(* CODESYS project Codesys_ADT
   Author: Riley Duffy
   Company: Bosch Rexroth
   DefaultNamespace: ADT
   Description: Abstract Data Type Framework
   Title: ADT
   Version: 1.0.0

Project tree, tasks and I/O mapping:
  libraries: Standard, 3.5.18.0 (System)
  BoschSE_ADT.Sync
  commdata.all
  DUT/
    data type DummyType
    data type HashData
    data type PVoid
  DynamicInterfaces (Not Yet Tested)/
    interface iDynamicDataContainer: CopyToNew, EndResize, GetNew, GetNewPointer, StartResize
    interface iDynamicHashTable: Clear, Delete, isDeleted, isNewOccupied, isOccupied
  function block GettingStarted [ST]
  Interfaces/
    interface iCompare: Compare
    interface iDataContainer: Get, GetPointer, GetSize, Put
    interface iHash: Hash
    interface iHashTable: Clear, Delete, isDeleted, isOccupied
    interface iIterable: GetIterator, isBusy
    interface iIterator: Next, Size
    interface iList: Clear, CloseIterator, Find, Get, GetIterator, GetPointer, Insert, Pop, PushFront, Put, Remove
    interface iMap: Clear, Get, HasKey, Put, Remove
    interface iQueue: PopFront, PushBack, Size
    interface iStack: PopBack, PushBack, Size
  libADT.Sync
  function block License_And_Use [ST]
  POUs/
    ResizableMem (Not Fully Tested)/
      function block DynamicHashTable [ST]: Clear, Compare, CopyToNew, Delete, EndResize, Get, GetNew, GetNewPointer, GetPointer, GetSize, Hash, isDeleted, isNewOccupied, isOccupied, Put, StartResize
      function block DynamicList [ST]: Clear, CloseIterator, Find, Get, GetIterator, GetPointer, Insert, isBusy, Pop, PopBack, PopFront, PushBack, PushFront, Put, Remove, Resize, Size
      function block DynamicMap [ST]: Clear, Get, HasKey, Put, Remove, Resize
      function block DynamicQueue [ST]: PopFront, PushBack, Resize, Size
    StaticMem/
      function block HashTable [ST]: Clear, Compare, Delete, Get, GetPointer, GetSize, Hash, isDeleted, isOccupied, Put
      function block Iterator [ST]: GetIterator, isBusy, Next, Size
      function block List [ST]: Clear, CloseIterator, Find, Get, GetIterator, GetPointer, Insert, isBusy, Pop, PopBack, PopFront, PushBack, PushFront, Put, Remove, Size
      function block Map [ST]: Clear, Get, HasKey, Put, Remove
      function block Queue [ST]: PopFront, PushBack, Size
    Templates/
      function block TemplateDynamicContainer [ST]: CopyToNew, EndResize, FB_Exit, FB_Init, Get, GetNew, GetNewPointer, GetPointer, GetSize, Put, StartResize
      function block TemplateStaticDataContainer [ST]: Get, GetPointer, GetSize, Put
    Util/
      function block ADT_CompareString [ST]: Compare
      function block StringHash [ST]: Hash
  function GetLibVersion [ST]
  function GetLibVersionNumber [ST]
  function IsLibReleased [ST]
  function GetBooleanProperty [ST]
  function GetCompany [ST]
  function GetTextProperty2 [ST]
  function GetTextProperty [ST]
  function GetTitle [ST]
  function GetVersion [ST]
  function GetVersionProperty [ST]
*)

// DUT/DummyType
TYPE DummyType :
STRUCT
	dummy : BOOL; 
END_STRUCT
END_TYPE

// DUT/HashData
{attribute 'enable_dynamic_creation'}
TYPE HashData :
STRUCT
	isOccupied : BOOL; 
	isDeleted  : BOOL; 
END_STRUCT
END_TYPE

// DUT/PVoid
TYPE PVoid : __XWORD; END_TYPE

// GettingStarted
(*Use the Template container in POUs/Templates to quickly create your ADT Container. 
  Edit the _size and the DummyType to the size and type you want*)


FUNCTION_BLOCK GettingStarted
VAR_INPUT
END_VAR
VAR_OUTPUT
END_VAR
VAR
END_VAR

END_FUNCTION_BLOCK

// License_And_Use
(*
Copyright  2025 Riley Duffy

Permission is hereby granted, free of charge, to any person obtaining a copy of this software and associated documentation files
the “Software”), to deal in the Software without restriction, including without limitation the rights to use, copy, modify, merge,
publish, distribute, sublicense, and/or sell copies of the Software, and to permit persons to whom the Software is furnished to do so,
subject to the following conditions:

The above copyright notice and this permission notice shall be included in all copies or substantial portions of the Software.

THE SOFTWARE IS PROVIDED “AS IS”, WITHOUT WARRANTY OF ANY KIND, EXPRESS OR IMPLIED,
 INCLUDING BUT NOT LIMITED TO THE WARRANTIES OF MERCHANTABILITY, FITNESS FOR A PARTICULAR PURPOSE AND NONINFRINGEMENT.
 IN NO EVENT SHALL THE AUTHORS OR COPYRIGHT HOLDERS BE LIABLE FOR ANY CLAIM, DAMAGES OR OTHER LIABILITY,
 WHETHER IN AN ACTION OF CONTRACT, TORT OR OTHERWISE, ARISING FROM, OUT OF OR IN CONNECTION WITH THE SOFTWARE
 OR THE USE OR OTHER DEALINGS IN THE SOFTWARE.*)
FUNCTION_BLOCK License_And_Use
VAR_INPUT
END_VAR
VAR_OUTPUT
END_VAR
VAR
END_VAR

(*
Copyright  2025 Riley DUffy

Permission is hereby granted, free of charge, to any person obtaining a copy of this software and associated documentation files
(the “Software”), to deal in the Software without restriction, including without limitation the rights to use, copy, modify, merge,
publish, distribute, sublicense, and/or sell copies of the Software, and to permit persons to whom the Software is furnished to do so,
subject to the following conditions:

The above copyright notice and this permission notice shall be included in all copies or substantial portions of the Software.

THE SOFTWARE IS PROVIDED “AS IS”, WITHOUT WARRANTY OF ANY KIND, EXPRESS OR IMPLIED,
 INCLUDING BUT NOT LIMITED TO THE WARRANTIES OF MERCHANTABILITY, FITNESS FOR A PARTICULAR PURPOSE AND NONINFRINGEMENT.
 IN NO EVENT SHALL THE AUTHORS OR COPYRIGHT HOLDERS BE LIABLE FOR ANY CLAIM, DAMAGES OR OTHER LIABILITY,
 WHETHER IN AN ACTION OF CONTRACT, TORT OR OTHERWISE, ARISING FROM, OUT OF OR IN CONNECTION WITH THE SOFTWARE
 OR THE USE OR OTHER DEALINGS IN THE SOFTWARE.*)

END_FUNCTION_BLOCK

// DynamicInterfaces (Not Yet Tested)/iDynamicDataContainer
INTERFACE iDynamicDataContainer Extends iDataContainer;

METHOD CopyToNew : BOOL
VAR_INPUT
	indexOld :UDINT; 
	indexNew :UDINT; 
END_VAR
END_METHOD

METHOD EndResize : BOOL
VAR_INPUT
END_VAR
END_METHOD

METHOD GetNew : BOOL
VAR_INPUT
	index : UDINT;
	pData : PVoid;  
END_VAR
END_METHOD

METHOD GetNewPointer : PVoid
VAR_INPUT
	index : UDINT;
END_VAR
END_METHOD

METHOD StartResize : BOOL
VAR_INPUT
END_VAR
END_METHOD

END_INTERFACE

// Interfaces/iDataContainer
INTERFACE iDataContainer

METHOD Get : Bool
VAR_INPUT
	index : UDINT;
	pData : PVoid;  
END_VAR
END_METHOD

METHOD GetPointer : PVoid
VAR_INPUT
	index : UDINT;
END_VAR
END_METHOD

METHOD GetSize : UDINT
VAR_INPUT
END_VAR
END_METHOD

METHOD Put : Bool
VAR_INPUT
	index : UDINT; 
	pData : PVoid; 
END_VAR
END_METHOD

END_INTERFACE

// DynamicInterfaces (Not Yet Tested)/iDynamicHashTable
INTERFACE iDynamicHashTable EXTENDS iDynamicDataContainer,iCompare,iHash

METHOD Clear : Bool
VAR_INPUT
END_VAR
END_METHOD

METHOD Delete : Bool
VAR_INPUT
	index : UDINT; 
END_VAR
END_METHOD

METHOD isDeleted : Bool
VAR_INPUT
	index : UDINT;
END_VAR
END_METHOD

METHOD isNewOccupied : BOOL
VAR_INPUT
	index : UDINT; 
END_VAR
END_METHOD

METHOD isOccupied : bool
VAR_INPUT
	index : UDINT; 
END_VAR
END_METHOD

END_INTERFACE

// Interfaces/iCompare
INTERFACE iCompare

METHOD Compare : INT
VAR_INPUT
	pData1 : PVoid; 
	pData2 : PVoid; 
END_VAR
END_METHOD

END_INTERFACE

// Interfaces/iHash
INTERFACE iHash

METHOD Hash : LINT
VAR_INPUT
	pData : pVoid; 
END_VAR
END_METHOD

END_INTERFACE

// Interfaces/iHashTable
INTERFACE iHashTable EXTENDS iDataContainer,iCompare,iHash

METHOD Clear : Bool
VAR_INPUT
END_VAR
END_METHOD

METHOD Delete : Bool
VAR_INPUT
	index : UDINT; 
END_VAR
END_METHOD

METHOD isDeleted : Bool
VAR_INPUT
	index : UDINT;
END_VAR
END_METHOD

METHOD isOccupied : bool
VAR_INPUT
	index : UDINT; 
END_VAR
END_METHOD

END_INTERFACE

// Interfaces/iIterable
INTERFACE iIterable

METHOD GetIterator : iIterator
VAR_INPUT
END_VAR
END_METHOD

PROPERTY isBusy : BOOL
GET
END_GET
END_PROPERTY

END_INTERFACE

// Interfaces/iIterator
INTERFACE iIterator EXTENDS iIterable

METHOD Next : BOOL
VAR_INPUT
	pData : PVOID; 
END_VAR
END_METHOD

PROPERTY Size : UDINT
GET
END_GET
END_PROPERTY

END_INTERFACE

// Interfaces/iList
INTERFACE iList EXTENDS iStack,iQueue,iIterable

METHOD Clear : BOOL
VAR_INPUT
END_VAR
END_METHOD

METHOD CloseIterator : BOOL
VAR_INPUT
END_VAR
END_METHOD

METHOD Find : iIterator
VAR_INPUT
	Where : iCompare; 
	pData : PVoid; 
	indexList : iList;
END_VAR
END_METHOD

METHOD Get : BOOL
VAR_INPUT
	Index : UDINT; 
	pData : PVOID; 
END_VAR
END_METHOD

METHOD GetIterator : iIterator
VAR_INPUT
	
END_VAR
END_METHOD

METHOD GetPointer : Bool
VAR_INPUT
	Index	: UDINT;
END_VAR
VAR_OUTPUT
	pData : PVoid; 
END_VAR
END_METHOD

METHOD Insert : BOOL
VAR_INPUT
	StartIndex : UDINT; 
	Values   : iIterable; 
END_VAR
END_METHOD

METHOD Pop : BOOL
VAR_INPUT
	Index : UDINT; 
	pData : PVOID; 
END_VAR
END_METHOD

METHOD PushFront : BOOL
VAR_INPUT
	pData : PVOID; 
END_VAR
END_METHOD

METHOD Put : BOOL
VAR_INPUT
	Index : UDINT; 
	pData : PVoid; 
END_VAR
END_METHOD

METHOD Remove : BOOL
VAR_INPUT
	Where : iCompare; 
	pData : PVoid; 
END_VAR
END_METHOD

END_INTERFACE

// Interfaces/iStack
INTERFACE iStack

METHOD PopBack : Bool
VAR_INPUT
	pData : PVoid; 
END_VAR
END_METHOD

METHOD PushBack : Bool
VAR_INPUT
	pData : PVOID; 
END_VAR
END_METHOD

PROPERTY Size : UDINT
GET
END_GET
END_PROPERTY

END_INTERFACE

// Interfaces/iQueue
INTERFACE iQueue

METHOD PopFront : Bool
VAR_INPUT
	pData : PVoid; 
END_VAR
END_METHOD

METHOD PushBack : Bool
VAR_INPUT
	pData : PVOID; 
END_VAR
END_METHOD

PROPERTY Size : UDINT
GET
END_GET
END_PROPERTY

END_INTERFACE

// Interfaces/iMap
INTERFACE iMap

METHOD Clear : Bool
VAR_INPUT
END_VAR
END_METHOD

METHOD Get : Bool
VAR_INPUT
	pKey : pVoid; 
	pValue : pVoid; 
END_VAR
END_METHOD

METHOD HasKey : Bool
VAR_INPUT
	pKey : pVoid; 
END_VAR
END_METHOD

METHOD Put : Bool
VAR_INPUT
	pKey : pVoid; 
	pValue : pVoid; 
END_VAR
END_METHOD

METHOD Remove : Bool
VAR_INPUT
	pKey : pVoid; 
END_VAR
END_METHOD

END_INTERFACE

// GetLibVersion
// This function has been automatically generated from the project information.
FUNCTION GetLibVersion : VERSION
VAR_INPUT
	
END_VAR

GetLibVersion.uiMajor := 1;
GetLibVersion.uiMinor := 0;
GetLibVersion.uiServicePack := 0;
GetLibVersion.uiPatch := 65535;

END_FUNCTION

// GetLibVersionNumber
// This function has been automatically generated from the project information.
FUNCTION GetLibVersionNumber : DWORD
VAR_INPUT
	
END_VAR

GetLibVersionNumber := 16777471;

END_FUNCTION

// IsLibReleased
// This function has been automatically generated from the project information.
FUNCTION IsLibReleased : BOOL
VAR_INPUT
	
END_VAR

IsLibReleased := FALSE;

END_FUNCTION

// GetBooleanProperty
// This function has been automatically generated from the project information.
{attribute 'signature_flag' := '1073741824'}
{attribute 'register_in_runtime'}
FUNCTION GetBooleanProperty : BOOL
VAR_INPUT
	stKey: WSTRING;
END_VAR

IF stKey = "Released" THEN
	GetBooleanProperty := FALSE;
ELSE
	GetBooleanProperty := FALSE;
END_IF

END_FUNCTION

// GetCompany
// This function has been automatically generated from the project information.
{attribute 'signature_flag' := '1073741824'}
{attribute 'register_in_runtime'}
FUNCTION GetCompany : WSTRING
VAR_INPUT
	
END_VAR

GetCompany := "Bosch Rexroth";

END_FUNCTION

// GetTextProperty2
// This function has been automatically generated from the project information.
{attribute 'signature_flag' := '1073741824'}
{attribute 'register_in_runtime'}
FUNCTION GetTextProperty2 : POINTER TO WSTRING
VAR_INPUT
	stKey: WSTRING;
END_VAR

IF stKey = "Author" THEN
	GetTextProperty2 := ADR("Riley Duffy");
ELSIF stKey = "Company" THEN
	GetTextProperty2 := ADR("Bosch Rexroth");
ELSIF stKey = "DefaultNamespace" THEN
	GetTextProperty2 := ADR("ADT");
ELSIF stKey = "Description" THEN
	GetTextProperty2 := ADR("Abstract Data Type Framework");
ELSIF stKey = "Project" THEN
	GetTextProperty2 := ADR("BoschSE_ADT");
ELSIF stKey = "Title" THEN
	GetTextProperty2 := ADR("ADT");
ELSE
	GetTextProperty2 := ADR("");
END_IF

END_FUNCTION

// GetTextProperty
// This function has been automatically generated from the project information.
{attribute 'signature_flag' := '1073741824'}
{attribute 'register_in_runtime'}
FUNCTION GetTextProperty : WSTRING
VAR_INPUT
	stKey: WSTRING;
END_VAR

IF stKey = "Author" THEN
	GetTextProperty := "Riley Duffy";
ELSIF stKey = "Company" THEN
	GetTextProperty := "Bosch Rexroth";
ELSIF stKey = "DefaultNamespace" THEN
	GetTextProperty := "ADT";
ELSIF stKey = "Description" THEN
	GetTextProperty := "Abstract Data Type Framework";
ELSIF stKey = "Project" THEN
	GetTextProperty := "BoschSE_ADT";
ELSIF stKey = "Title" THEN
	GetTextProperty := "ADT";
ELSE
	GetTextProperty := "";
END_IF

END_FUNCTION

// GetTitle
// This function has been automatically generated from the project information.
{attribute 'signature_flag' := '1073741824'}
{attribute 'register_in_runtime'}
FUNCTION GetTitle : WSTRING
VAR_INPUT
	
END_VAR

GetTitle := "ADT";

END_FUNCTION

// GetVersion
// This function has been automatically generated from the project information.
{attribute 'signature_flag' := '1073741824'}
{attribute 'register_in_runtime'}
FUNCTION GetVersion : VERSION
VAR_INPUT
	
END_VAR

GetVersion.uiMajor := 1;
GetVersion.uiMinor := 0;
GetVersion.uiServicePack := 0;
GetVersion.uiPatch := 65535;

END_FUNCTION

// GetVersionProperty
// This function has been automatically generated from the project information.
{attribute 'signature_flag' := '1073741824'}
{attribute 'register_in_runtime'}
FUNCTION GetVersionProperty : VERSION
VAR_INPUT
	stKey: WSTRING;
END_VAR

IF stKey = "Version" THEN
	GetVersionProperty.uiMajor := 1;
	GetVersionProperty.uiMinor := 0;
	GetVersionProperty.uiServicePack := 0;
	GetVersionProperty.uiPatch := 65535;
ELSE
	GetVersionProperty.uiMajor := 0;
	GetVersionProperty.uiMinor := 0;
	GetVersionProperty.uiServicePack := 0;
	GetVersionProperty.uiPatch := 0;
END_IF

END_FUNCTION

// POUs/ResizableMem (Not Fully Tested)/DynamicHashTable
{attribute 'no_check'}
FUNCTION_BLOCK DynamicHashTable IMPLEMENTS iDynamicHashTable
VAR_INPUT
	KeyContainer : iDynamicDataContainer;
	HashDataContainer : iDynamicDataContainer;  
	Compareator : iCompare;
	Hasher      : iHash;  
END_VAR
VAR_OUTPUT
END_VAR
VAR
END_VAR

{attribute 'no_check'}
METHOD Clear : BOOL
VAR
	tHashData : HashData; 
	i : UDINT; 
END_VAR
tHashData.isDeleted := FALSE; 
tHashData.isOccupied := FALSE; 
FOR i := 0 TO HashDataContainer.GetSize() DO 
	HashDataContainer.Put(i,ADR(tHashData)); 
END_FOR
END_METHOD

METHOD Compare : INT
VAR_INPUT
	pData1	: PVoid;
	pData2	: PVoid;
END_VAR
Compare := Compareator.Compare(pData1,pData2);
END_METHOD

METHOD CopyToNew : BOOL
VAR_INPUT
	indexOld	: UDINT;
	indexNew	: UDINT;
END_VAR
KeyContainer.CopyToNew(indexOld,indexNew);
HashDataContainer.CopyToNew(indexOld,indexNew);
END_METHOD

METHOD Delete : BOOL
VAR_INPUT
	index	: UDINT;
END_VAR
VAR
	tHashData : HashData; 
END_VAR
tHashData.isDeleted := TRUE; 
tHashData.isOccupied := FALSE; 
HashDataContainer.Put(index,ADR(tHashData));
END_METHOD

METHOD EndResize : BOOL
KeyContainer.StartResize(); 
HashDataContainer.StartResize();
END_METHOD

METHOD Get : BOOL
VAR_INPUT
	index	: UDINT;
	pData	: PVoid;
END_VAR
KeyContainer.Get(index,pData);
END_METHOD

METHOD GetNew : BOOL
VAR_INPUT
	index : UDINT;
	pData : PVoid;  
END_VAR
KeyContainer.GetNew(index,pData);
END_METHOD

METHOD GetNewPointer : PVoid
VAR_INPUT
	index	: UDINT;
END_VAR
GetNewPointer := KeyContainer.GetNewPointer(index);
END_METHOD

METHOD GetPointer : PVoid
VAR_INPUT
	index	: UDINT;
END_VAR
GetPointer := KeyContainer.GetPointer(index);
END_METHOD

METHOD GetSize : UDINT
GetSize := KeyContainer.GetSize();
END_METHOD

METHOD Hash : LINT
VAR_INPUT
	pData	: pVoid;
END_VAR
Hash := Hasher.Hash(pData);
END_METHOD

METHOD isDeleted : BOOL
VAR_INPUT
	index	: UDINT;
END_VAR
VAR
	tHashData : HashData; 
END_VAR
HashDataContainer.Get(index,ADR(tHashData)); 
isDeleted := tHashData.isDeleted;
END_METHOD

METHOD isNewOccupied : BOOL
VAR_INPUT
	index: UDINT;
END_VAR
VAR
	tHashData: HashData;
END_VAR
HashDataContainer.GetNew(index,ADR(tHashData)); 
isNewOccupied:= tHashData.isOccupied;
END_METHOD

METHOD isOccupied : BOOL
VAR_INPUT
	index	: UDINT;
END_VAR
VAR
	tHashData : HashData; 
END_VAR
HashDataContainer.Get(index,ADR(tHashData)); 
isOccupied:= tHashData.isOccupied;
END_METHOD

METHOD Put : BOOL
VAR_INPUT
	index	: UDINT;
	pData	: PVoid;
END_VAR
VAR
	tHashData : HashData; 
END_VAR
tHashData.isDeleted := FALSE; 
tHashData.isOccupied := TRUE; 
HashDataContainer.Put(index,ADR(tHashData)); 
KeyContainer.Put(index,pData);
END_METHOD

METHOD StartResize : BOOL
KeyContainer.StartResize(); 
HashDataContainer.StartResize();
END_METHOD

END_FUNCTION_BLOCK

// POUs/ResizableMem (Not Fully Tested)/DynamicList
{attribute 'no_check'}
FUNCTION_BLOCK DynamicList IMPLEMENTS iList
VAR_INPUT
	DataContainer :  iDynamicDataContainer; 
END_VAR
VAR_OUTPUT
END_VAR
VAR
	_size : UDINT; 
	_iterator : Iterator; 
	_bIteratorOpened : BOOL; 
	_backingSize: UDINT;
	_front: UDINT;
END_VAR

METHOD Clear : BOOL
_size := 0;
END_METHOD

METHOD CloseIterator : BOOL
_bIteratorOpened := FALSE;
END_METHOD

{attribute 'no_check'}
METHOD Find : iIterator
VAR_INPUT
	Where	: iCompare;
	pData	: PVoid;
	indexList	: iList;
END_VAR
VAR
	_i : UDINT; 
	_index : UDINT; 
END_VAR
IF _backingSize = 0 THEN 
	_backingSize := DataContainer.GetSize(); 
END_IF
IF NOT _bIteratorOpened THEN 
	indexList.Clear(); 
	FOR _i := 0 TO _size -1 DO 
		IF Where.Compare(pData,DataContainer.GetPointer((_i + _front) MOD _backingSize)) = 0 THEN 
			_index := (_i + _front)MOD _backingSize; 
			indexList.PushBack(ADR(_index)); 
		END_IF
	END_FOR
	_iterator(bAll := FALSE, 
		  refList := THIS^, 
		  refIndex := indexList);
	Find := _iterator; 
	_bIteratorOpened := TRUE; 
ELSE
	Find := _iterator; 
END_IF;
END_METHOD

METHOD Get : BOOL
VAR_INPUT
	Index	: UDINT;
	pData	: PVOID;
END_VAR
IF _backingSize = 0 THEN 
	_backingSize := DataContainer.GetSize(); 
END_IF
IF Index < _size THEN 
	Get := DataContainer.Get((Index + _front) MOD _backingSize ,pData); 
ELSE 
	Get := FALSE; 
END_IF
END_METHOD

METHOD GetIterator : iIterator
IF NOT _bIteratorOpened THEN
	_bIteratorOpened := TRUE;  
	_iterator(bAll := TRUE, 
			refList := THIS^
			);
	GetIterator := _iterator; 
ELSE 
	GetIterator := _iterator; 
END_IF
END_METHOD

METHOD GetPointer : Bool
VAR_INPUT
	Index	: UDINT;
END_VAR
VAR_OUTPUT
	pData : PVoid; 
END_VAR
IF _backingSize = 0 THEN 
	_backingSize := DataContainer.GetSize(); 
END_IF
IF Index < _size THEN 
	pData := DataContainer.GetPointer((Index + _front) MOD _backingSize);
	GetPointer := TRUE; 
ELSE 
	GetPointer := FALSE; 
END_IF
END_METHOD

METHOD Insert : BOOL
VAR_INPUT
	StartIndex	: UDINT; //Start Index
	Values	: iIterable; //Iterable list of values to insert
END_VAR

VAR
	_i: UDINT;
	_index: UDINT;
	_destIndex: UDINT;
END_VAR
IF _backingSize = 0 THEN 
	_backingSize := DataContainer.GetSize(); 
END_IF
WHILE Values.GetIterator().Size >= (_backingSize - size) DO 
	_backingSize := THIS^.Resize();
END_WHILE
IF StartIndex <= _size AND NOT Values.GetIterator().isBusy THEN 
	IF StartIndex <> _size THEN 
		FOR _i := _size - 1  TO StartIndex BY - 1 DO
			_index := (_front + _i) MOD _backingSize; 
			_destIndex := (_index + Values.GetIterator().Size) MOD _backingSize; 
			DataContainer.Put(_destIndex,DataContainer.GetNewPointer(_index)); 
			IF _i = 0 THEN 
				EXIT; 
			END_IF
		END_FOR
	END_IF
	WHILE Values.GetIterator().Next(DataContainer.GetPointer((StartIndex + _front + _i) MOD _backingSize)) DO 
		_i := _i+1; 
		_size := _size + 1; 
	END_WHILE
	Insert := TRUE; 
ELSE 
	Insert := FALSE; 
END_IF
END_METHOD

PROPERTY isBusy : BOOL
GET
isBusy := _bIteratorOpened;
END_GET
END_PROPERTY

METHOD Pop : BOOL
VAR_INPUT
	Index	: UDINT;
	pData	: PVOID;
END_VAR

VAR
	_i: UDINT;
	_index: UDINT;
	_indexPlus1: UDINT;
END_VAR
IF _backingSize = 0 THEN 
	_backingSize := DataContainer.GetSize(); 
END_IF
IF Index < _size THEN 
	Pop := DataContainer.Get((Index + _front) MOD _backingSize,pData); 
	FOR _i := Index TO size -1 DO 
		_index := (_front + _i) MOD _backingSize; 
		_indexPlus1 := (_index + 1) MOD _backingSize; 
		DataContainer.Put(_index,DataContainer.GetPointer(_indexPlus1)); 
		IF _i = 0 THEN 
			EXIT; 
		END_IF
	END_FOR
	_size := _size - 1; 
ELSE 
	Pop := FALSE; 
END_IF
END_METHOD

METHOD PopBack : BOOL
VAR_INPUT
	pData	: PVoid;
END_VAR

VAR
END_VAR
IF _backingSize = 0 THEN 
	_backingSize := DataContainer.GetSize(); 
END_IF
IF _size > 0 THEN 
	PopBack := DataContainer.Get((_front + _size) MOD _backingSize ,pData); 
	_size := _size - 1; 
ELSE 
	PopBack := FALSE; 
END_IF
END_METHOD

METHOD PopFront : BOOL
VAR_INPUT
	pData	: PVoid;
END_VAR
IF _backingSize = 0 THEN 
	_backingSize := DataContainer.GetSize(); 
END_IF
IF _size > 0 THEN 
	PopFront := DataContainer.Get(_front,pData); 
	_size := _size - 1; 
	_front := (_front + 1) MOD _backingSize; 
ELSE 
	PopFront := FALSE; 
END_IF
END_METHOD

METHOD PushBack : BOOL
VAR_INPUT
	pData	: PVOID;
END_VAR
IF _backingSize = 0 THEN 
	_backingSize := DataContainer.GetSize(); 
END_IF
IF _size >= _backingSize THEN 
	_backingSize := THIS^.Resize(); 
END_IF
IF _size < _backingSize THEN 
	PushBack := DataContainer.Put((_front+_size) MOD _backingSize,pData); 
	_size := _size + 1;
ELSE 
	PushBack := FALSE; 
END_IF
END_METHOD

METHOD PushFront : BOOL
VAR_INPUT
	pData	: PVOID;
END_VAR
IF _backingSize = 0 THEN 
	_backingSize := DataContainer.GetSize(); 
END_IF
IF _size >= _backingSize THEN 
	_backingSize := THIS^.Resize(); 
END_IF
IF _size < _backingSize THEN 
	_front := _front -1; 
	IF _front >= _backingSize THEN 
		_front := _backingSize - 1; 
	END_IF
	PushFront := DataContainer.Put(_front,pData); 
	_size := _size + 1; 
ELSE 
	PushFront := FALSE; 
END_IF
END_METHOD

METHOD Put : BOOL
VAR_INPUT
	Index	: UDINT;
	pData	: PVoid;
END_VAR

VAR
	_i: UDINT;
	_index : UDINT;
	_indexSub1 : UDINT; 
END_VAR
IF _backingSize = 0 THEN 
	_backingSize := DataContainer.GetSize(); 
END_IF
IF _size >= _backingSize THEN 
	_backingSize := THIS^.Resize(); 
END_IF
IF _size < _backingSize AND Index <= _size THEN 
	IF Index <> _size THEN 
		FOR _i := _size  TO Index + 1 BY - 1 DO
			_index := (_front + _i) MOD _backingSize; 
			_indexSub1 := _index - 1; 
			IF (_indexSub1 >= _backingSize) THEN 
				_indexSub1 := _backingSize -1; 
			END_IF
			DataContainer.Put(_index,DataContainer.GetPointer(_indexSub1)); 
		END_FOR
	END_IF
	Put := DataContainer.Put((Index + _front)MOD _backingSize,pData); 
	_size := _size + 1; 
ELSE 
	Put := FALSE; 
END_IF
END_METHOD

METHOD Remove : BOOL
VAR_INPUT
	Where	: iCompare;
	pData   : PVoid; 
END_VAR

VAR
	_i: UDINT;
	_j: UDINT;
	_index : UDINT; 
	_indexPlus1 : UDINT; 
END_VAR
Remove := FALSE; 
IF _size = 0 THEN 
	RETURN; 
END_IF
FOR _i := 0 TO _size -1 DO 
	IF Where.Compare(pData,DataContainer.GetPointer((_i + _front) MOD _backingSize)) = 0 THEN 
		FOR _j := _i  TO _size-1 DO 
			_index := (_front + _j) MOD _backingSize; 
			_indexPlus1 := (_index + 1) MOD _backingSize; 
			DataContainer.Put(_index,DataContainer.GetPointer(_indexPlus1)); 
		END_FOR
		_size := _size - 1; 
		Remove := TRUE; 
		EXIT; 
	END_IF;
END_FOR
END_METHOD

METHOD PRIVATE Resize : UDINT
VAR_INPUT
END_VAR

VAR
	_i: UDINT;
END_VAR
DataContainer.StartResize(); 
FOR _i := 0 TO THIS^.Size -1 DO 
	DataContainer.CopyToNew((_front + _i) MOD _backingSize, _i); 
END_FOR
_front := 0; 
DataContainer.EndResize();
Resize := DataContainer.GetSize();
END_METHOD

PROPERTY Size : UDINT
GET
Size := _size;
END_GET
END_PROPERTY

END_FUNCTION_BLOCK

// POUs/StaticMem/Iterator
FUNCTION_BLOCK Iterator IMPLEMENTS iIterator
VAR_INPUT
	bAll : BOOL; 
	refList : iList; 
	refIndex :  iList; 
END_VAR
VAR_OUTPUT
END_VAR
VAR
	_index : UDINT; 
END_VAR

_index := 0;

METHOD GetIterator : iIterator
GetIterator := This^;
END_METHOD

PROPERTY isBusy : BOOL
GET
isBusy := _index <> 0;
END_GET
END_PROPERTY

{attribute 'no_check'}
METHOD Next : BOOL
VAR_INPUT
	pData	: PVOID;
END_VAR
VAR 
	pIndex : UDINT; 
END_VAR
IF bAll THEN 
	IF _index <refList.Size THEN 
		IF refList.Get(_index ,pData) THEN 
			_index := _index + 1; 
			Next := TRUE; 
		ELSE 
			_index := 0; 
			refList.CloseIterator(); 
			Next := FALSE; 
		END_IF
	ELSE 
		_index := 0; 
		refList.CloseIterator(); 
		Next := FALSE; 
	END_IF
ELSE 
	IF _index < refIndex.Size THEN 
		IF refIndex.Get(_index,ADR(pIndex)) THEN 
			refList.Get(pIndex,pData); 
			_index := _index + 1; 
			Next := TRUE; 
		ELSE 
			_index := 0; 
			refIndex.Clear(); 
			refList.CloseIterator(); 
			Next := FALSE; 
		END_IF
	ELSE 
		_index := 0; 
		refList.CloseIterator(); 
		Next := FALSE; 
	END_IF	
END_IF
END_METHOD

PROPERTY Size : UDINT
GET
IF bAll THEN 
	Size := refList.Size;
ELSE
	Size := refIndex.Size;
END_IF
END_GET
END_PROPERTY

END_FUNCTION_BLOCK

// POUs/StaticMem/List
{attribute 'no_check'}
FUNCTION_BLOCK List IMPLEMENTS iList
VAR_INPUT
	DataContainer : iDataContainer; 
END_VAR
VAR_OUTPUT
END_VAR
VAR
	_size : UDINT; 
	_iterator : Iterator; 
	_bIteratorOpened : BOOL; 
	_backingSize: UDINT;
	_front: UDINT;
END_VAR

METHOD Clear : BOOL
_size := 0;
END_METHOD

METHOD CloseIterator : BOOL
_bIteratorOpened := FALSE;
END_METHOD

{attribute 'no_check'}
METHOD Find : iIterator
VAR_INPUT
	Where	: iCompare;
	pData	: PVoid;
	indexList	: iList;
END_VAR
VAR
	_i : UDINT; 
	_index : UDINT; 
END_VAR
IF _backingSize = 0 THEN 
	_backingSize := DataContainer.GetSize(); 
END_IF
IF NOT _bIteratorOpened THEN 
	indexList.Clear(); 
	FOR _i := 0 TO _size -1 DO 
		IF Where.Compare(pData,DataContainer.GetPointer((_i + _front) MOD _backingSize)) = 0 THEN 
			_index := (_i + _front)MOD _backingSize; 
			indexList.PushBack(ADR(_index)); 
		END_IF
	END_FOR
	_iterator(bAll := FALSE, 
		  refList := THIS^, 
		  refIndex := indexList);
	Find := _iterator; 
	_bIteratorOpened := TRUE; 
ELSE
	Find := _iterator; 
END_IF;
END_METHOD

METHOD Get : BOOL
VAR_INPUT
	Index	: UDINT;
	pData	: PVOID;
END_VAR
IF _backingSize = 0 THEN 
	_backingSize := DataContainer.GetSize(); 
END_IF
IF Index < _size THEN 
	Get := DataContainer.Get((Index + _front) MOD _backingSize ,pData); 
ELSE 
	Get := FALSE; 
END_IF
END_METHOD

METHOD GetIterator : iIterator
IF NOT _bIteratorOpened THEN
	_bIteratorOpened := TRUE;  
	_iterator(bAll := TRUE, 
			refList := THIS^
			);
	GetIterator := _iterator; 
ELSE 
	GetIterator := _iterator; 
END_IF
END_METHOD

METHOD GetPointer : Bool
VAR_INPUT
	Index	: UDINT;
END_VAR
VAR_OUTPUT
	pData : PVoid; 
END_VAR
IF _backingSize = 0 THEN 
	_backingSize := DataContainer.GetSize(); 
END_IF
IF Index < _size THEN 
	pData := DataContainer.GetPointer((Index + _front) MOD _backingSize);
	GetPointer := TRUE; 
ELSE 
	GetPointer := FALSE; 
END_IF
END_METHOD

METHOD Insert : BOOL
VAR_INPUT
	StartIndex	: UDINT; //Index Insertion Starts At
	Values	: iIterable; //Iterable list of values to insert
END_VAR

VAR
	_i: UDINT;
	_index: UDINT;
	_destIndex: UDINT;
END_VAR
IF _backingSize = 0 THEN 
	_backingSize := DataContainer.GetSize(); 
END_IF
IF Values.GetIterator().Size < (_backingSize - size) AND StartIndex <= _size AND NOT Values.GetIterator().isBusy THEN 
	IF StartIndex <> _size THEN 
		FOR _i := _size - 1  TO StartIndex BY - 1 DO
			_index := (_front + _i) MOD _backingSize; 
			_destIndex := (_index + Values.GetIterator().Size) MOD _backingSize; 
			DataContainer.Put(_destIndex,DataContainer.GetPointer(_index)); 
			IF _i = 0 THEN 
				EXIT; 
			END_IF
		END_FOR
	END_IF
	WHILE Values.GetIterator().Next(DataContainer.GetPointer((StartIndex + _front + _i) MOD _backingSize)) DO 
		_i := _i+1; 
		_size := _size + 1; 
	END_WHILE
	Insert := TRUE; 
ELSE 
	Insert := FALSE; 
END_IF
END_METHOD

PROPERTY isBusy : BOOL
GET
isBusy := _bIteratorOpened;
END_GET
END_PROPERTY

METHOD Pop : BOOL
VAR_INPUT
	Index	: UDINT;
	pData	: PVOID;
END_VAR

VAR
	_i: UDINT;
	_index: UDINT;
	_indexPlus1: UDINT;
END_VAR
IF _backingSize = 0 THEN 
	_backingSize := DataContainer.GetSize(); 
END_IF
IF Index < _size THEN 
	Pop := DataContainer.Get((Index + _front) MOD _backingSize,pData); 
	FOR _i := Index TO size -1 DO 
		_index := (_front + _i) MOD _backingSize; 
		_indexPlus1 := (_index + 1) MOD _backingSize; 
		DataContainer.Put(_index,DataContainer.GetPointer(_indexPlus1)); 
		IF _i = 0 THEN 
			EXIT; 
		END_IF
	END_FOR
	_size := _size - 1; 
ELSE 
	Pop := FALSE; 
END_IF
END_METHOD

METHOD PopBack : BOOL
VAR_INPUT
	pData	: PVoid;
END_VAR

VAR
END_VAR
IF _backingSize = 0 THEN 
	_backingSize := DataContainer.GetSize(); 
END_IF
IF _size > 0 THEN 
	PopBack := DataContainer.Get((_front + _size) MOD _backingSize ,pData); 
	_size := _size - 1; 
ELSE 
	PopBack := FALSE; 
END_IF
END_METHOD

METHOD PopFront : BOOL
VAR_INPUT
	pData	: PVoid;
END_VAR
IF _backingSize = 0 THEN 
	_backingSize := DataContainer.GetSize(); 
END_IF
IF _size > 0 THEN 
	PopFront := DataContainer.Get(_front,pData); 
	_size := _size - 1; 
	_front := (_front + 1) MOD _backingSize; 
ELSE 
	PopFront := FALSE; 
END_IF
END_METHOD

METHOD PushBack : BOOL
VAR_INPUT
	pData	: PVOID;
END_VAR
IF _backingSize = 0 THEN 
	_backingSize := DataContainer.GetSize(); 
END_IF
IF _size < _backingSize THEN 
	PushBack := DataContainer.Put((_front+_size) MOD _backingSize,pData); 
	_size := _size + 1; 
ELSE 
	PushBack := FALSE; 
END_IF
END_METHOD

METHOD PushFront : BOOL
VAR_INPUT
	pData	: PVOID;
END_VAR
IF _backingSize = 0 THEN 
	_backingSize := DataContainer.GetSize(); 
END_IF
IF _size < _backingSize THEN 
	_front := _front -1; 
	IF _front >= _backingSize THEN 
		_front := _backingSize - 1; 
	END_IF
	PushFront := DataContainer.Put(_front,pData); 
	_size := _size + 1; 
ELSE 
	PushFront := FALSE; 
END_IF
END_METHOD

METHOD Put : BOOL
VAR_INPUT
	Index	: UDINT;
	pData	: PVoid;
END_VAR

VAR
	_i: UDINT;
	_index : UDINT;
	_indexSub1 : UDINT; 
END_VAR
IF _backingSize = 0 THEN 
	_backingSize := DataContainer.GetSize(); 
END_IF
IF _size < _backingSize AND Index <= _size THEN 
	IF Index <> _size THEN 
		FOR _i := _size  TO Index + 1 BY - 1 DO
			_index := (_front + _i) MOD _backingSize; 
			_indexSub1 := _index - 1; 
			IF (_indexSub1 >= _backingSize) THEN 
				_indexSub1 := _backingSize -1; 
			END_IF
			DataContainer.Put(_index,DataContainer.GetPointer(_indexSub1)); 
		END_FOR
	END_IF
	Put := DataContainer.Put((Index + _front)MOD _backingSize,pData); 
	_size := _size + 1; 
ELSE 
	Put := FALSE; 
END_IF
END_METHOD

METHOD Remove : BOOL
VAR_INPUT
	Where	: iCompare;
	pData   : PVoid; 
END_VAR

VAR
	_i: UDINT;
	_j: UDINT;
	_index : UDINT; 
	_indexPlus1 : UDINT; 
END_VAR
Remove := FALSE; 
IF _size = 0 THEN 
	RETURN; 
END_IF
FOR _i := 0 TO _size -1 DO 
	IF Where.Compare(pData,DataContainer.GetPointer((_i + _front) MOD _backingSize)) = 0 THEN 
		FOR _j := _i  TO _size-1 DO 
			_index := (_front + _j) MOD _backingSize; 
			_indexPlus1 := (_index + 1) MOD _backingSize; 
			DataContainer.Put(_index,DataContainer.GetPointer(_indexPlus1)); 
		END_FOR
		_size := _size - 1; 
		Remove := TRUE; 
		EXIT; 
	END_IF;
END_FOR
END_METHOD

PROPERTY Size : UDINT
GET
Size := _size;
END_GET
END_PROPERTY

END_FUNCTION_BLOCK

// POUs/ResizableMem (Not Fully Tested)/DynamicMap
{attribute 'no_check'}
FUNCTION_BLOCK DynamicMap IMPLEMENTS iMap
VAR_INPUT
	KeyContainer : iDynamicHashTable; 
	ValueContainer : iDynamicDataContainer; 
END_VAR
VAR_OUTPUT
END_VAR
VAR
	_backingSize : UDINT := 0;
	_size : DINT := 0;  
END_VAR

METHOD Clear : BOOL
KeyContainer.Clear();
END_METHOD

{attribute 'no_check'}
METHOD Get : BOOL
VAR_INPUT
	pKey	: pVoid;
	pValue	: pVoid;
END_VAR

VAR
	hash: LINT;
	index: UDINT;
	_i : UDINT; 
	_tIndex: UDINT;
END_VAR
Get := FALSE; 
IF(_backingSize = 0 ) THEN 
	_backingSize := KeyContainer.GetSize(); 
END_IF
hash :=  KeyContainer.Hash(pKey); 
index := LINT_TO_UDINT(hash MOD _backingSize); 
WHILE _i < _backingSize - 1 DO 
	_tIndex := (_i + index) MOD _backingSize; 
	IF NOT (KeyContainer.isOccupied(_tIndex) OR KeyContainer.isDeleted(_tIndex))THEN 
		EXIT; 
	END_IF
	IF KeyContainer.Compare(pKey, KeyContainer.GetPointer(_tIndex)) = 0 THEN 
		ValueContainer.Get(_tIndex,pValue); 
		Get := TRUE; 
		EXIT; 
	END_IF
	_i := _i+ 1; 
END_WHILE
END_METHOD

{attribute 'no_check'}
METHOD HasKey : BOOL
VAR_INPUT
	pKey : pVoid; 
END_VAR

VAR
	hash: LINT;
	index: UDINT;
	_i: UDINT;
	_tIndex: UDINT;
END_VAR
HasKey := FALSE; 
IF(_backingSize = 0 ) THEN 
	_backingSize := KeyContainer.GetSize(); 
END_IF
hash :=  KeyContainer.Hash(pKey); 
index := LINT_TO_UDINT(hash MOD _backingSize); 
WHILE _i < _backingSize - 1 DO 
	_tIndex := (_i + index) MOD _backingSize; 
	IF NOT (KeyContainer.isOccupied(_tIndex) OR KeyContainer.isDeleted(_tIndex))THEN 
		EXIT; 
	END_IF
	IF KeyContainer.Compare(pKey, KeyContainer.GetNewPointer(_tIndex)) = 0 THEN  
		HasKey := TRUE; 
		EXIT; 
	END_IF
	_i := _i+ 1; 
END_WHILE
END_METHOD

{attribute 'no_check'}
METHOD Put : BOOL
VAR_INPUT
	pKey	: pVoid;
	pValue	: pVoid;
END_VAR

VAR
	hash: LINT;
	index: UDINT;
	_i: UDINT;
	_tIndex: UDINT;
END_VAR
Put := FALSE; 
IF(_backingSize = 0 ) THEN 
	_backingSize := KeyContainer.GetSize(); 
END_IF
IF _size >= _backingSize THEN 
	_backingSize := resize(); 
END_IF
hash :=  KeyContainer.Hash(pKey); 
index := LINT_TO_UDINT(hash MOD _backingSize); 
WHILE _i < _backingSize - 1 DO 
	_tIndex := (_i + index) MOD _backingSize; 
	IF (KeyContainer.isOccupied(_tIndex)) THEN 
		IF KeyContainer.Compare(pKey, KeyContainer.GetNewPointer(_tIndex)) = 0 THEN 
			ValueContainer.Put(_tIndex,pValue); 
			PUT := TRUE; 
			EXIT;
		END_IF
	ELSE 
		ValueContainer.Put(_tIndex,pValue); 
		KeyContainer.Put(_tIndex,pKey); 
		PUT := TRUE; 
		_size := _size + 1; 
		EXIT;
	END_IF 	
	_i := _i + 1; 
END_WHILE
END_METHOD

{attribute 'no_check'}
METHOD Remove : BOOL
VAR_INPUT
	pKey	: pVoid;
END_VAR

VAR
	hash: LINT;
	index: UDINT;
	_i: UDINT;
	_tIndex: UDINT;
END_VAR
Remove := FALSE; 
IF(_backingSize = 0 ) THEN 
	_backingSize := KeyContainer.GetSize(); 
END_IF
hash :=  KeyContainer.Hash(pKey); 
index := LINT_TO_UDINT(hash MOD _backingSize); 
WHILE _i < _backingSize - 1 DO 
	_tIndex := (_i + index) MOD _backingSize; 
	IF NOT (KeyContainer.isOccupied(_tIndex) OR KeyContainer.isDeleted(_tIndex))THEN 
		EXIT; 
	END_IF
	IF KeyContainer.Compare(pKey, KeyContainer.GetNewPointer(_tIndex)) = 0 THEN 
		KeyContainer.Delete(_tIndex);  
		Remove := TRUE; 
		_size := _size -1; 
		EXIT; 
	END_IF
	_i := _i+ 1; 
END_WHILE
END_METHOD

METHOD PRIVATE Resize : UDINT
VAR_INPUT
END_VAR

VAR
	_i: UDINT;
	_newSize: UDINT;
	index: UDINT;
	hash: LINT;
	_tIndex: UDINT;
	_j: UINT;
END_VAR
ValueContainer.StartResize();
KeyContainer.StartResize(); 
_newSize := KeyContainer.GetSize(); 
FOR _i := 0 TO _backingSize DO 
	IF KeyContainer.isOccupied(_i) THEN 
		hash :=  KeyContainer.Hash(KeyContainer.GetPointer(_i)); 
		index := LINT_TO_UDINT(hash MOD _newSize); 
		_j := 0; 
		WHILE _j < _backingSize - 1 DO 
			_tIndex := (_j + index) MOD _newSize; 
			IF (KeyContainer.isNewOccupied(_tIndex)) THEN 
				IF KeyContainer.Compare(KeyContainer.GetPointer(_i), KeyContainer.GetNewPointer(_tIndex)) = 0 THEN 
					KeyContainer.CopyToNew(_i,_tindex); 
					ValueContainer.CopyToNew(_i,_tindex); 
					EXIT;
				END_IF
			ELSE 
				KeyContainer.CopyToNew(_i,_tindex); 
				ValueContainer.CopyToNew(_i,_tindex); 
				EXIT;
			END_IF 	
			_j := _j + 1; 
		END_WHILE
	END_IF
END_FOR
Resize := 2*_backingSize; 
ValueContainer.EndResize();
KeyContainer.EndResize();
END_METHOD

END_FUNCTION_BLOCK

// POUs/ResizableMem (Not Fully Tested)/DynamicQueue
{attribute 'no_check'}
FUNCTION_BLOCK DynamicQueue IMPLEMENTS iQueue
VAR_INPUT
	DataContainer : iDynamicDataContainer; 
END_VAR
VAR_OUTPUT
END_VAR
VAR
	_size : UDINT; 
	_front: UDINT; 
	_backingSize : UDINT := 0; 
END_VAR

METHOD PopFront : BOOL
VAR_INPUT
	pData: PVoid;
END_VAR
IF _backingSize = 0 THEN 
	_backingSize := DataContainer.GetSize(); 
END_IF
IF _size > 0 THEN 
	PopFront := DataContainer.Get(_front,pData); 
	_size := _size - 1; 
	_front := (_front + 1) MOD _backingSize; 
ELSE 
	PopFront := FALSE; 
END_IF
END_METHOD

METHOD PushBack : BOOL
VAR_INPUT
	pData : pVoid; 
END_VAR
IF _backingSize = 0 THEN 
	_backingSize := DataContainer.GetSize(); 
END_IF
IF _size = _backingSize THEN 
	_backingSize := resize(); 
END_IF
IF _size < _backingSize THEN 
	PushBack := DataContainer.Put((_front+_size) MOD _backingSize,pData); 
	_size := _size + 1; 
ELSE 
	PushBack := FALSE; 
END_IF
END_METHOD

METHOD PRIVATE Resize : UDINT
VAR_INPUT
END_VAR

VAR
	_i: UDINT;
END_VAR
DataContainer.StartResize(); 
FOR _i := 0 TO THIS^.Size DO 
	DataContainer.CopyToNew((_front + _i) MOD _size, _i); 
END_FOR
_front := 0; 
DataContainer.EndResize();
Resize := DataContainer.GetSize();
END_METHOD

PROPERTY Size : UDINT
GET
Size := _size;
END_GET
END_PROPERTY

END_FUNCTION_BLOCK

// POUs/StaticMem/HashTable
{attribute 'no_check'}
FUNCTION_BLOCK HashTable IMPLEMENTS iHashTable
VAR_INPUT
	KeyContainer : iDataContainer;
	HashDataContainer : iDataContainer;  
	Compareator : iCompare;
	Hasher      : iHash;  
END_VAR
VAR_OUTPUT
END_VAR
VAR
END_VAR

{attribute 'no_check'}
METHOD Clear : BOOL
VAR
	tHashData : HashData; 
	i : UDINT; 
END_VAR
tHashData.isDeleted := FALSE; 
tHashData.isOccupied := FALSE; 
FOR i := 0 TO HashDataContainer.GetSize() DO 
	HashDataContainer.Put(i,ADR(tHashData)); 
END_FOR
END_METHOD

METHOD Compare : INT
VAR_INPUT
	pData1	: PVoid;
	pData2	: PVoid;
END_VAR
Compare := Compareator.Compare(pData1,pData2);
END_METHOD

METHOD Delete : BOOL
VAR_INPUT
	index	: UDINT;
END_VAR
VAR
	tHashData : HashData; 
END_VAR
tHashData.isDeleted := TRUE; 
tHashData.isOccupied := FALSE; 
HashDataContainer.Put(index,ADR(tHashData));
END_METHOD

METHOD Get : BOOL
VAR_INPUT
	index	: UDINT;
	pData	: PVoid;
END_VAR
KeyContainer.Get(index,pData);
END_METHOD

METHOD GetPointer : PVoid
VAR_INPUT
	index	: UDINT;
END_VAR
GetPointer := KeyContainer.GetPointer(index);
END_METHOD

METHOD GetSize : UDINT
GetSize := KeyContainer.GetSize();
END_METHOD

METHOD Hash : LINT
VAR_INPUT
	pData	: pVoid;
END_VAR
Hash := Hasher.Hash(pData);
END_METHOD

METHOD isDeleted : BOOL
VAR_INPUT
	index	: UDINT;
END_VAR
VAR
	tHashData : HashData; 
END_VAR
HashDataContainer.Get(index,ADR(tHashData)); 
isDeleted := tHashData.isDeleted;
END_METHOD

METHOD isOccupied : BOOL
VAR_INPUT
	index	: UDINT;
END_VAR
VAR
	tHashData : HashData; 
END_VAR
HashDataContainer.Get(index,ADR(tHashData)); 
isOccupied:= tHashData.isOccupied;
END_METHOD

METHOD Put : BOOL
VAR_INPUT
	index	: UDINT;
	pData	: PVoid;
END_VAR
VAR
	tHashData : HashData; 
END_VAR
tHashData.isDeleted := FALSE; 
tHashData.isOccupied := TRUE; 
HashDataContainer.Put(index,ADR(tHashData)); 
KeyContainer.Put(index,pData);
END_METHOD

END_FUNCTION_BLOCK

// POUs/StaticMem/Map
{attribute 'no_check'}
FUNCTION_BLOCK Map IMPLEMENTS iMap
VAR_INPUT
	KeyContainer : iHashTable; 
	ValueContainer : iDataContainer; 
END_VAR
VAR_OUTPUT
END_VAR
VAR
	_backingSize : UDINT := 0; 
END_VAR

METHOD Clear : BOOL
KeyContainer.Clear();
END_METHOD

{attribute 'no_check'}
METHOD Get : BOOL
VAR_INPUT
	pKey	: pVoid;
	pValue	: pVoid;
END_VAR

VAR
	hash: LINT;
	index: UDINT;
	_i : UDINT; 
	_tIndex: UDINT;
END_VAR
Get := FALSE; 
IF(_backingSize = 0 ) THEN 
	_backingSize := KeyContainer.GetSize(); 
END_IF
hash :=  KeyContainer.Hash(pKey); 
index := LINT_TO_UDINT(hash MOD _backingSize); 
WHILE _i < _backingSize - 1 DO 
	_tIndex := (_i + index) MOD _backingSize; 
	IF NOT (KeyContainer.isOccupied(_tIndex) OR KeyContainer.isDeleted(_tIndex))THEN 
		EXIT; 
	END_IF
	IF KeyContainer.Compare(pKey, KeyContainer.GetPointer(_tIndex)) = 0 THEN 
		ValueContainer.Get(_tIndex,pValue); 
		Get := TRUE; 
		EXIT; 
	END_IF
	_i := _i+ 1; 
END_WHILE
END_METHOD

{attribute 'no_check'}
METHOD HasKey : BOOL
VAR_INPUT
	pKey : pVoid; 
END_VAR

VAR
	hash: LINT;
	index: UDINT;
	_i: UDINT;
	_tIndex: UDINT;
END_VAR
HasKey := FALSE; 
IF(_backingSize = 0 ) THEN 
	_backingSize := KeyContainer.GetSize(); 
END_IF
hash :=  KeyContainer.Hash(pKey); 
index := LINT_TO_UDINT(hash MOD _backingSize); 
WHILE _i < _backingSize - 1 DO 
	_tIndex := (_i + index) MOD _backingSize; 
	IF NOT (KeyContainer.isOccupied(_tIndex) OR KeyContainer.isDeleted(_tIndex))THEN 
		EXIT; 
	END_IF
	IF KeyContainer.Compare(pKey, KeyContainer.GetPointer(_tIndex)) = 0 THEN  
		HasKey := TRUE; 
		EXIT; 
	END_IF
	_i := _i+ 1; 
END_WHILE
END_METHOD

{attribute 'no_check'}
METHOD Put : BOOL
VAR_INPUT
	pKey	: pVoid;
	pValue	: pVoid;
END_VAR

VAR
	hash: LINT;
	index: UDINT;
	_i: UDINT;
	_tIndex: UDINT;
END_VAR
Put := FALSE; 
IF(_backingSize = 0 ) THEN 
	_backingSize := KeyContainer.GetSize(); 
END_IF
hash :=  KeyContainer.Hash(pKey); 
index := LINT_TO_UDINT(hash MOD _backingSize); 
WHILE _i < _backingSize - 1 DO 
	_tIndex := (_i + index) MOD _backingSize; 
	IF (KeyContainer.isOccupied(_tIndex)) THEN 
		IF KeyContainer.Compare(pKey, KeyContainer.GetPointer(_tIndex)) = 0 THEN 
			ValueContainer.Put(_tIndex,pValue); 
			PUT := TRUE; 
			EXIT;
		END_IF
	ELSE 
		ValueContainer.Put(_tIndex,pValue); 
		KeyContainer.Put(_tIndex,pKey); 
		PUT := TRUE; 
		EXIT;
	END_IF 	
	_i := _i + 1; 
END_WHILE
END_METHOD

{attribute 'no_check'}
METHOD Remove : BOOL
VAR_INPUT
	pKey	: pVoid;
END_VAR

VAR
	hash: LINT;
	index: UDINT;
	_i: UDINT;
	_tIndex: UDINT;
END_VAR
Remove := FALSE; 
IF(_backingSize = 0 ) THEN 
	_backingSize := KeyContainer.GetSize(); 
END_IF
hash :=  KeyContainer.Hash(pKey); 
index := LINT_TO_UDINT(hash MOD _backingSize); 
WHILE _i < _backingSize - 1 DO 
	_tIndex := (_i + index) MOD _backingSize; 
	IF NOT (KeyContainer.isOccupied(_tIndex) OR KeyContainer.isDeleted(_tIndex))THEN 
		EXIT; 
	END_IF
	IF KeyContainer.Compare(pKey, KeyContainer.GetPointer(_tIndex)) = 0 THEN 
		KeyContainer.Delete(_tIndex);  
		Remove := TRUE; 
		EXIT; 
	END_IF
	_i := _i+ 1; 
END_WHILE
END_METHOD

END_FUNCTION_BLOCK

// POUs/StaticMem/Queue
{attribute 'no_check'}
FUNCTION_BLOCK Queue IMPLEMENTS iQueue
VAR_INPUT
	DataContainer : iDataContainer; 
END_VAR
VAR_OUTPUT
END_VAR
VAR
	_size : UDINT; 
	_front: UDINT; 
	_backingSize : UDINT := 0; 
END_VAR

METHOD PopFront : BOOL
VAR_INPUT
	pData: PVoid;
END_VAR
IF _backingSize = 0 THEN 
	_backingSize := DataContainer.GetSize(); 
END_IF
IF _size > 0 THEN 
	PopFront := DataContainer.Get(_front,pData); 
	_size := _size - 1; 
	_front := (_front + 1) MOD _backingSize; 
ELSE 
	PopFront := FALSE; 
END_IF
END_METHOD

METHOD PushBack : BOOL
VAR_INPUT
	pData : pVoid; 
END_VAR
IF _backingSize = 0 THEN 
	_backingSize := DataContainer.GetSize(); 
END_IF
IF _size < _backingSize THEN 
	PushBack := DataContainer.Put((_front+_size) MOD _backingSize,pData); 
	_size := _size + 1; 
ELSE 
	PushBack := FALSE; 
END_IF
END_METHOD

PROPERTY Size : UDINT
GET
Size := _size;
END_GET
END_PROPERTY

END_FUNCTION_BLOCK

// POUs/Templates/TemplateDynamicContainer
FUNCTION_BLOCK TemplateDynamicContainer IMPLEMENTS iDynamicDataContainer
VAR_INPUT
	udSize : UDINT; 
END_VAR
VAR_OUTPUT
END_VAR
VAR
	_ptrBackingArray : POINTER TO DummyType;
	_ptrTempNewArray : POINTER TO DummyType;  
	_size : UDINT; 
	_tData : DummyType; 
	_pData : POINTER TO DummyType; 
	_newSize: UDINT;
	_byteSize : UDINT; 
END_VAR

_byteSize := SIZEOF(_tData); 
_newSize := udSize * _byteSize;
_ptrBackingArray := __NEW(BYTE,_newSize); 
_size := udSize;

METHOD CopyToNew : BOOL
VAR_INPUT
	indexOld	: UDINT;
	indexNew	: UDINT;
END_VAR
CopyToNew := FALSE; 
IF indexOld < _size/2 AND indexNew < _size THEN 
	_ptrTempNewArray[indexNew] := _ptrBackingArray[indexOld]; 
	CopyToNew := TRUE; 
END_IF
END_METHOD

METHOD EndResize : BOOL
__DELETE(_ptrBackingArray); 
_ptrBackingArray := _ptrTempNewArray; 
_ptrTempNewArray := 0;
END_METHOD

//FB_Exit must be implemented explicitly. If there is an implementation, then the
//method is called before the controller removes the code of the function block instance
//(implicit call). The return value is not evaluated.
METHOD FB_Exit: BOOL
VAR_INPUT
    bInCopyCode: BOOL;  // TRUE: the exit method is called in order to leave the instance which will be copied afterwards (online change).  
END_VAR
if _ptrBackingArray <> 0 THEN 
	__DELETE(_ptrBackingArray); 
END_IF
IF _ptrTempNewArray <> 0 THEN 
	__DELETE(_ptrTempNewArray); 
END_IF
END_METHOD

//FB_Init is always available implicitly and it is used primarily for initialization.
//The return value is not evaluated. For a specific influence, you can also declare the
//methods explicitly and provide additional code there with the standard initialization
//code. You can evaluate the return value.
METHOD FB_Init: BOOL
VAR_INPUT
    bInitRetains: BOOL; // TRUE: the retain variables are initialized (reset warm / reset cold)
    bInCopyCode: BOOL;  // TRUE: the instance will be copied to the copy code afterward (online change) 
	udSize      : UDINT;   
END_VAR
this^(udSize := udSize);
END_METHOD

METHOD Get : BOOL
VAR_INPUT
	index	: UDINT;
	pData	: PVoid;
END_VAR
IF index < _size THEN 
	_pData := pData; 
	_pData^ := _ptrBackingArray[index]; 
	GET := TRUE; 
ELSE 
	GET := FALSE; 
END_IF
END_METHOD

METHOD GetNew : BOOL
VAR_INPUT
	index	: UDINT;
	pData	: PVoid;
END_VAR
IF _ptrTempNewArray <> 0 AND index < _size THEN 
	_pData := pData; 
	_pData^ :=_ptrTempNewArray[index]; 
	GetNew := TRUE; 
ELSE 
	GetNew := FALSE; 
END_IF
END_METHOD

METHOD GetNewPointer : PVoid
VAR_INPUT
	index	: UDINT;
END_VAR
IF _ptrTempNewArray <> 0 AND index < _size THEN 
	GetNewPointer := ADR(_ptrTempNewArray[index]); 
ELSE 
	GetNewPointer := 0; 
END_IF
END_METHOD

METHOD GetPointer : PVoid
VAR_INPUT
	index	: UDINT;
END_VAR
IF index < _size THEN 
	GetPointer := ADR(_ptrBackingArray[index]); 
ELSE 
	GetPointer := 0; 
END_IF
END_METHOD

METHOD GetSize : UDINT
GetSize :=_size;
END_METHOD

METHOD Put : BOOL
VAR_INPUT
	index	: UDINT;
	pData	: PVoid;
END_VAR
_pData := pData; 
Put := FALSE; 
IF index < _size THEN 
	_ptrBackingArray[index] := _pData^; 
	Put := TRUE; 
END_IF
END_METHOD

METHOD StartResize : BOOL
VAR
	_newSize: UDINT;
END_VAR
_newSize := (2* _size)*_byteSize;
_ptrTempNewArray := __NEW(BYTE,_newSize); 
_size := _size * 2;
END_METHOD

END_FUNCTION_BLOCK

// POUs/Templates/TemplateStaticDataContainer
{attribute 'no_check'}
FUNCTION_BLOCK TemplateStaticDataContainer IMPLEMENTS iDataContainer
VAR_INPUT
	
END_VAR
VAR_OUTPUT
END_VAR
VAR CONSTANT
	_size : UDINT := 100; 
END_VAR 
VAR
	_arBacking : ARRAY[0.._size - 1] OF DummyType;
	_pData : POINTER TO DummyType;
END_VAR

{attribute 'no_check'}
METHOD Get : BOOL
VAR_INPUT
	index	: UDINT;
	pData	: PVoid;
END_VAR
_pData := pData; 
IF index < _size THEN 
	_pData^ := _arBacking[index]; 
	Get := TRUE;
ELSE 
	Get := FALSE; 
END_IF
END_METHOD

{attribute 'no_check'}
METHOD GetPointer : PVoid
VAR_INPUT
	index	: UDINT;
END_VAR
IF index < _size THEN 
	GetPointer:= ADR(_arBacking[index]); 
ELSE 
	GetPointer := 0; 
END_IF
END_METHOD

METHOD GetSize : UDINT
GetSize := _size;
END_METHOD

{attribute 'no_check'}
METHOD Put : BOOL
VAR_INPUT
	index	: UDINT;
	pData	: PVoid;
END_VAR
_pData := pData; 
IF index < _size THEN 
	_arBacking[index] := _pData^; 
	Put := TRUE; 
ELSE 
	Put := FALSE; 
END_IF
END_METHOD

END_FUNCTION_BLOCK

// POUs/Util/ADT_CompareString
FUNCTION_BLOCK ADT_CompareString Implements iCompare
VAR_INPUT
END_VAR
VAR_OUTPUT
END_VAR
VAR
END_VAR

{warning 'Add method implementation '}
(* Pointers to the data being comapred are passed, 
   Compare >0 Data1 > Data2 
   Compare <0 Data1 < Data2 
   Compare = 0 Data 1 = Data2 *)
METHOD Compare : INT
VAR_INPUT
	pData1	: PVoid;
	pData2	: PVoid;
END_VAR
VAR
	pString1 : POINTER TO STRING := pData1; 
	pString2 : POINTER TO STRING := pData2; 
END_VAR
IF pString1^ = pString2^ THEN 
	Compare := 0; 
	RETURN;
END_IF
Compare := 1;
END_METHOD

END_FUNCTION_BLOCK

// POUs/Util/StringHash
{attribute 'no_check'}
FUNCTION_BLOCK StringHash IMPLEMENTS iHash
VAR_INPUT
END_VAR
VAR_OUTPUT
END_VAR
VAR
END_VAR

{attribute 'no_check'}
METHOD Hash : LINT
VAR_INPUT
	pData	: pVoid;
END_VAR
VAR
	ptrString : POINTER TO String := pData; 
	_i: INT;
	_multiple: LINT;
	_hash : LINT; 
END_VAR
_multiple := 1; 
_hash := 0; 
FOR _i :=0 TO LEN(ptrString^) - 1 DO 
	_hash := _hash + ptrString^[_i] * _multiple; 
	_multiple := _multiple + 1; 
END_FOR
Hash := _hash;
END_METHOD

END_FUNCTION_BLOCK
